FUNCTION CheckBounds : DINT
VAR_INPUT
    i, l, u : DINT;
END_VAR

IF i<l THEN
    CheckBounds := l;
ELSIF i>u THEN
    CheckBounds := u;
ELSE
    CheckBounds := i;
END_IF

END_FUNCTION

(* stored: Version 1.1.0.1, ProductVersion 3.1.4024.12
   POU CheckBounds: Id {729a14d1-dcc8-4f5b-8117-a8e6274e4f04}, SpecialFunc None *)
